					IF eMoverAccessoryID = MoverAccessoryID.APM9001_0000 THEN
						// Note: With the current driver release (3.2209.36.0) mover identification only works if all movers are equiped with ID bumpers!
						bWithBumperID := TRUE;						
					END_IF
				END_FOR
			END_FOR
		END_IF

			
		IF bWithBumperID THEN
			nStatePreparation := nStatePreparation + 10;
		ELSE
			nStatePreparation := 500;
		END_IF
		
	
	60: // 6th: Do mover identification
		//ipVisuMessage.SetInfoMessage('Start mover-identification', 'MoverPreparation', nStatePreparation);
	
		IF NOT bDeterminedMoverID THEN
			IF fbXPlanarSystem.UtilityCheckForError(bAutoReset := TRUE) > 0 THEN
// 				IF fbXPlanarSystem.ipDriver.TcIoXpu(1).SetCoordMoverCommunicationCmd(CoordinatedMoverCommCommand.IdentifyAndAssignPossible) THEN
				IF fbXPlanarSystem.ipDriver.TcIoXpu(1).SetCoordMoverCommunicationCmd(CoordinatedMoverCommCommand.IdentifyBTNsAndRearrangeMovers) THEN
					nStatePreparation := nStatePreparation +1;
				END_IF	
			END_IF
		ELSE
			nStatePreparation := nStatePreparation +10;
		END_IF
	
	61:
		IF fbXPlanarSystem.UtilityCheckForError(bAutoReset := TRUE) > 0 THEN			
			moverCoordComStatus := fbXPlanarSystem.ipDriver.TcIoXpu(1).GetCoordMoverCommStatus();
			
			IF moverCoordComStatus = CoordinatedMoverCommStatus.CommunicationSuccessful THEN
				bDeterminedMoverID := TRUE;
				//ipVisuMessage.ClearAllMessages();
				nStatePreparation := nStatePreparation + 4;
			ELSIF moverCoordComStatus = CoordinatedMoverCommStatus.CommunicationFailed THEN
				nStatePreparation := nStatePreparation + 1;	
			END_IF
			
		END_IF
		
	62:	IF fbXPlanarSystem.UtilityCheckForError(bAutoReset := TRUE) > 0 THEN	
			nMoverID_ErrorCode := fbXPlanarSystem.ipDriver.TcIoXpu(1).GetCoordMoverCommunicationErrorId();
			//ipVisuMessage.SetErrorMessage('Mover Identification Failed!', 'MoverPreparation', nStatePreparation, nMoverID_ErrorCode);
		END_IF
		
		//IF ipVisuMessage.CheckAknowledge()  THEN
		nStatePreparation := 0;	
		//END_IF
	
	65: 
		FOR idx:=1 TO GVL.g_nMoverCount DO
			fbMover[idx].P_MoverID := fbXPlanarSystem.ipDriver.TcIoXpu(1).TcIoMover(UDINT_TO_UINT(idx)).GetIdentifiedMoverBtn();
		END_FOR
		nStatePreparation := nStatePreparation + 5;
	70: // 7th: Determine Mover-Orientation
	
		// Note: At the time of creation of this example code only APM4330 was able to determine its orientation.
		//       Change the code according to newer driver releases and availability of the orientation feature.
		bMoverCanDeterminOrientation := TRUE;
		FOR idx:=1 TO GVL.g_nMoverCount DO
			MoverType := fbXPlanarSystem.ipDriver.TcIoXpu(1).TcIoMover(UDINT_TO_UINT(idx)).GetMoverType();
			IF MoverType <> XPlanarMoverType.APM4330 THEN
				bMoverCanDeterminOrientation := FALSE;
			END_IF
		END_FOR
			
		IF bMoverCanDeterminOrientation THEN
			IF NOT bDerterminedMoverOrientation THEN
				//ipVisuMessage.SetInfoMessage('Mover orientation determination', 'MoverPreparation', nStatePreparation);
				IF fbXPlanarSystem.UtilityCheckForError(bAutoReset := TRUE) > 0 THEN
					IF fbXPlanarSystem.ipDriver.TcIoXpu(1).SetCoordMoverCommunicationCmd(CoordinatedMoverCommCommand.DetermineOrientations) THEN
						nStatePreparation := nStatePreparation + 1;	
					END_IF
				END_IF
			ELSE
				nStatePreparation := nStatePreparation + 20;		
			END_IF
		ELSE
			nStatePreparation := nStatePreparation + 20;
		END_IF
	
		
	71: // Check if communication is active
		IF fbXPlanarSystem.UtilityCheckForError(bAutoReset := TRUE) > 0 THEN
			moverCoordComStatus := fbXPlanarSystem.ipDriver.TcIoXpu(1).GetCoordMoverCommStatus();
			IF moverCoordComStatus = CoordinatedMoverCommStatus.CommunicationInProcess THEN
				nStatePreparation := nStatePreparation + 1;	
			END_IF
		END_IF
	
		
	72: // Wait for orientation determination finished
		IF fbXPlanarSystem.UtilityCheckForError(bAutoReset := TRUE) > 0 THEN
			moverCoordComStatus := fbXPlanarSystem.ipDriver.TcIoXpu(1).GetCoordMoverCommStatus();
			IF moverCoordComStatus = CoordinatedMoverCommStatus.CommunicationSuccessful THEN
				nStatePreparation := nStatePreparation + 8;	
			ELSIF moverCoordComStatus = CoordinatedMoverCommStatus.CommunicationFailed THEN
				IF nCommunicationRetryCounter <= 5 THEN
					nCommunicationRetryCounter := nCommunicationRetryCounter +1;
					nStatePreparation := nStatePreparation - 2;	
				ELSE
					nStatePreparation := nStatePreparation + 1;	
				END_IF
			END_IF
		END_IF
		
				
	73:	// Check which movers do not communicate correctly:
		nMoverToCheck := 0;
		nStatePreparation := nStatePreparation + 1;
		
	74: nMoverToCheck := nMoverToCheck +1;
		IF nMoverToCheck <= GVL.g_nMoverCount THEN
			IF fbXPlanarSystem.UtilityCheckForError(bAutoReset := TRUE) > 0 THEN
				IF fbXPlanarSystem.ipDriver.TcIoXpu(1).TcIoMover(nMoverToCheck).SetMoverCommunicationCommand(MoverCommunicationCommand.DetermineOrientation) THEN
					nStatePreparation := nStatePreparation + 1;
				END_IF
			END_IF
		ELSE
			FOR idx:=1 TO GVL.g_nMoverCount DO
				bCommunicationProblem := FALSE;
				IF bMoverCommunicationProblem[idx] THEN
					bCommunicationProblem := TRUE;	
				END_IF
			END_FOR
			
			IF bCommunicationProblem THEN
				sTextTemp := 'Mover Communication Problem: ';
				FOR idx:=1 TO GVL.g_nMoverCount DO
					IF bMoverCommunicationProblem[idx] THEN
						sTextTemp := CONCAT(sTextTemp, ' M');
						sTextTemp := CONCAT(sTextTemp, UDINT_TO_STRING(idx));
					END_IF
				END_FOR				
				//ipVisuMessage.SetErrorMessage(sTextTemp, sTextTemp, nStatePreparation, 0);
			ELSE
				nStatePreparation := nStatePreparation - 4;	
			END_IF
		END_IF
		
	75: moverComStatus := fbXPlanarSystem.ipDriver.TcIoXpu(1).TcIoMover(nMoverToCheck).GetCommunicationStatus();
		IF moverComStatus = MoverCommunicationStatus.CommunicationSuccessful THEN
			bMoverCommunicationProblem[nMoverToCheck] := FALSE;
			nStatePreparation := nStatePreparation - 1;
		ELSIF moverComStatus = MoverCommunicationStatus.CommunicationFailed THEN
			bMoverCommunicationProblem[nMoverToCheck] := TRUE;
			nStatePreparation := nStatePreparation - 1;
		END_IF
		
		
	80:	// Rotation-Angle modulo adaption
		//ipVisuMessage.SetInfoMessage('Rotation-Angle modulo adaption', 'MoverPreparation', nStatePreparation);
		nMoverToCorrect := 0;
		nStatePreparation := nStatePreparation + 1;	
		
	81:	nMoverToCorrect := nMoverToCorrect +1;
		IF nMoverToCorrect <= GVL.g_nMoverCount THEN
			fMoverOrientationRead    := GVL.g_Movers[nMoverToCorrect].std.P_ActPosition.c; 
			fMoverOrientationCorrect := fMoverOrientationRead;
			 bDoRotationCorrection := FALSE;
			nStatePreparation := nStatePreparation + 1;	
		ELSE
			bDerterminedMoverOrientation := TRUE;
			nStatePreparation := nStatePreparation + 9;	
		END_IF
		
	82:	IF fMoverOrientationCorrect >= 0 THEN
			IF fMoverOrientationCorrect > 360.0 THEN
				fMoverOrientationCorrect := fMoverOrientationCorrect - 180.0;
				bDoRotationCorrection := TRUE;
			ELSE
				nStatePreparation := nStatePreparation + 1;
			END_IF
		ELSE
			IF fMoverOrientationCorrect < 360.0 THEN
				fMoverOrientationCorrect := fMoverOrientationCorrect + 180.0;
				bDoRotationCorrection := TRUE;
			ELSE
				nStatePreparation := nStatePreparation + 1;
			END_IF
		END_IF			
		
		
	83:	IF bDoRotationCorrection THEN
			
			fPosX := GVL.g_Movers[nMoverToCorrect].std.P_ActPosition.x;
			fPosY := GVL.g_Movers[nMoverToCorrect].std.P_ActPosition.y;
			fPosC := GVL.g_Movers[nMoverToCorrect].std.P_ActPosition.c;
	
			CorrectionPos.SetValuesXYC(fPosX, fPosY, fMoverOrientationCorrect);	
	
			GVL.g_Movers[nMoverToCorrect].std.SetMoverPosition('Correction', CorrectionPos);
			
			nStatePreparation := nStatePreparation + 1;	
		ELSE
			nStatePreparation := nStatePreparation - 2;
		END_IF
		
	84:
		IF GVL.g_Movers[nMoverToCorrect].std.P_SetMoverPosition.Done THEN
			nStatePreparation := nStatePreparation - 3;
		ELSIF GVL.g_Movers[nMoverToCorrect].std.P_SetMoverPosition.Error THEN
			nErrorID := GVL.g_Movers[nMoverToCorrect].std.P_SetMoverPosition.ErrorID;
			//ipVisuMessage.SetErrorMessage('Rotation-Angle modulo adaption', 'MoverPreparation', nStatePreparation, nErrorID);		
		END_IF
		

	90: nStatePreparation := 500;
	
			
	500: // Done
	//	nStatePreparation := 0;
		MoverPreparation := TRUE;		
			
		
	END_CASE


	//ipVisuMessage.StateUpdate(nStatePreparation, 'MoverPreparation');
END_METHOD

METHOD MoverRecovery : BOOL
VAR_INPUT
	bReset : BOOL;
END_VAR

VAR
	index : UDINT;
	ipMoverApplication: INT;
END_VAR

VAR_INST
	
	stOptionsJoinTrack				: ST_JoinTrackOptions;
	bMoversJoined 					: BOOL;
	bMoverError 					: BOOL;
	bMoverOrientationSet			: BOOL;
	bClearStation 					:ARRAY [1..GVL.gc_NumberStations] OF BOOL;
	bStationCleared					:bool;
	nMoverToTurn					: UDINT;
	nMoverToTurnBack				: UDINT;
	nTrackToCheck					:UDINT; 
	nDistanceToTrack				:LREAL;
	nDistanceToTargetTrack			: ARRAY[1..moverCount] OF REAL;
	nTargetTrack					: ARRAY[1..moverCount] OF UDINT;
	
	
	
	fRecoveryRotTarget				: LREAL;
	fRecoveryRotVel					: LREAL :=  360.0;
	fRecoveryRotAcc					: LREAL := 1800.0;
	fRecoveryRotJerk				: LREAL := 9000.0;
	stRotationOptions				: ST_MoveCOptions;




	
END_VAR
IF bReset THEN
	MoverRecovery := FALSE;
	nRecoverySequence := 0;
END_IF

CASE nRecoverySequence OF
	0:
		bMoversJoined := FALSE;
		bMoverError := FALSE;
		nMoverToTurn := 0;
		IF NOT bReset THEN
			nRecoverySequence := nRecoverySequence + 1;
		END_IF
		
	1: 	//set rotary orienation 
	
		FOR index := 1 TO gvl.g_nMoverCount DO
		fbXPlanarMover[index].MoveA('', 0, 100, 1000, 1000, 10000);
		fbXPlanarMover[index].MoveB('', 0, 100, 1000, 1000, 10000);
 		fbXPlanarMover[index].MoveC('', 0, 180, 1800, 1800, 18000, 0);
		
		END_FOR

		nRecoverySequence := nRecoverySequence + 1;
	
	2: 
		bMoverOrientationSet:= TRUE; 
		FOR index := 1 TO  gvl.g_nMoverCount DO
			IF fbXPlanarMover[index].P_MoveA.Done AND fbXPlanarMover[index].P_MoveB.Done AND fbXPlanarMover[index].P_MoveC.Done THEN 
				bMoverOrientationSet:= TRUE; 
			ELSE 
				bMoverOrientationSet:= FALSE; 
				
			END_IF
		END_FOR
		
		IF bMoverOrientationSet THEN
			nRecoverySequence := nRecoverySequence + 8;
	
		END_IF
	
	10:
	
		nMoverToTurn := nMoverToTurn +1;
		IF nMoverToTurn > gvl.g_nMoverCount THEN
				nRecoverySequence := nRecoverySequence +3;
			ELSE
				IF GVL.g_Movers[nMoverToTurn].std.P_IsPresent THEN

					fRecoveryRotTarget 				  := GVL.g_Movers[nMoverToTurn].std.P_ClosestQuaterAngle;	
					stRotationOptions.additionalTurns := 0;
					stRotationOptions.direction		  := Tc3_Mc3PlanarMotion.MC_direction.mcDirectionNonModulo;	
					
					GVL.g_Movers[nMoverToTurn].std.MoveC('Recovery - unfinished rotation', fRecoveryRotTarget, fRecoveryRotVel, fRecoveryRotAcc, fRecoveryRotAcc, fRecoveryRotJerk, stRotationOptions);
					nRecoverySequence := nRecoverySequence +1;				
				END_IF	
			END_IF
		
	
	11:
			IF GVL.g_Movers[nMoverToTurn].std.P_MoveC.Done THEN
				nRecoverySequence := nRecoverySequence -1;	
			ELSIF GVL.g_Movers[nMoverToTurn].std.P_MoveC.Error THEN
				nRecoverySequence := nRecoverySequence +1;	
			END_IF
			
	12: 		// Check error ID and react accordingly
			nErrorID := GVL.g_Movers[nMoverToTurn].std.P_MoveC.ErrorID;	
			
			// In case rotation is not possible due to collision with another mover proceed without rotation correction.
			IF nErrorID = 33158 THEN
				nRecoverySequence := nRecoverySequence -2;	
			END_IF

	13: 	nRecoverySequence := 100;	

		    
	100: 
			bStationCleared:=TRUE;
			bClearStation[GVL.PuncherStation]:=fbPuncherStation.Clear();
			bClearStation[GVL.PuncherSeparateStation]:=fbPuncherSeparateStation.Clear();
			bClearStation[GVL.PuncherBufferStation]:=fbPuncherBufferStation.Clear();
	
	FOR  index := 1 TO  GVL.gc_NumberStations DO
		IF bClearStation[index] THEN
			bStationCleared:=TRUE;
			ELSE
				bStationCleared:=FALSE;
		END_IF
	END_FOR
	IF bStationCleared THEN
			nRecoverySequence := 200;

		END_IF
		
// 	110: // look for for nearest track 
// 	
// 	
// 	FOR nMoverToTurnBack := 1 TO  gvl.g_nMoverCount DO
// 		nDistanceToTargetTrack[nMoverToTurnBack]:= 999999;
// 		
// 		FOR nTrackToCheck :=1 TO GVL.gc_NumberTracks DO 
// 		nDistanceToTrack := fbXPlanarMover[ nMoverToTurnBack].GetDistanceToTrack(GVL.g_Tracks[nTrackToCheck].std);
// 		
// 		IF nDistanceToTrack < nDistanceToTargetTrack[nMoverToTurnBack] AND nDistanceToTrack<> -1 THEN 
// 			nDistanceToTargetTrack[nMoverToTurnBack]:=nDistanceToTrack;
// 			nTargetTrack[nMoverToTurnBack] :=nTrackToCheck;
// 		END_IF
// 		
// 	END_FOR
// 	
// 	END_FOR
// 	
// 	nRecoverySequence := nRecoverySequence +10;
// 	
// 	120: // join to track
// 
// 		stOptionsJoinTrack.useOrientation := TRUE;
// 		
// 		FOR index := 1 TO gvl.g_nMoverCount DO
// 		IF fbXPlanarMover[index].P_CommandMode<> MC_PLANAR_MOVER_COMMAND_MODE.OnTrack THEN
// 			fbXPlanarMover[index].JoinTrack('Joining track', GVL.g_Tracks[nTargetTrack[index]].std, 250, 1250, 12500, stOptionsJoinTrack);
// 			
// 		END_IF
// 		
// 			
// END_FOR
// 	
// 		nRecoverySequence := nRecoverySequence + 1;
// 		
// 	121:
// 		bMoversJoined := TRUE;
// 		bMoverError := FALSE;
// 		FOR index := 1 TO moverCount DO
// 			bMoversJoined := bMoversJoined AND fbXPlanarMover[index].P_JoinTrack.Done;
// 			IF  fbXPlanarMover[index].P_JoinTrack.Done THEN 
// 				gvl.g_Movers[index].P_TrackId:=nTargetTrack[index];
// 			END_IF
// 			bMoverError := bMoverError OR fbXPlanarMover[index].P_JoinTrack.Error;			
// 		END_FOR
// 		
// 	IF bMoversJoined THEN
// 			nRecoverySequence := nRecoverySequence + 9;
// 	ELSIF bMoverError THEN
//  			nRecoverySequence := nRecoverySequence + 4;
// 	END_IF
// 		
		
// 	130: //send mover to station 
// 	  	  
// 		FOR index := 1 TO gvl.g_nMoverCount DO
// 			 IF fbXPlanarMover[index].P_TrackId= GVL.TrackPuncherWellplate THEN 
// 				 fbPuncherStation.P_List_Switch_Input_W.AddMover(GVL.g_Movers[index].std);
// 		
// 			
// 			 END_IF
// 		END_FOR
// 
// 		nRecoverySequence := 200;

	200: 
		MoverRecovery := TRUE;
		
END_CASE
END_METHOD

METHOD Resetting : BOOL
VAR_INPUT
END_VAR

VAR
	index : UDINT;
	MC_PLANNAR_: ST_CommandReturn;
END_VAR


VAR_INST
	
	nTrackToEnable		: UDINT;
	stProductDataClear 	: ST_ProductData;
	stOptionsJoinTrack				: ST_JoinTrackOptions;
	bMoversJoined 					: BOOL;
	bMoverError 					: BOOL;
	nMoverToTurn					: UDINT;
	nMoverToTurnBack				: UDINT;
	nTrackToCheck					:UDINT; 
	nDistanceToTrack				:LREAL;
	nDistanceToTargetTrack			: ARRAY[1..moverCount] OF REAL;
	nTargetTrack					: ARRAY[1..moverCount] OF UDINT;
	
END_VAR
nErrorID := 0;

CASE nResettingSequence OF 
	
	0: // Enter 
		nResettingSequence := 10;
		
		
		
	10: // Reset all movers
		IF fbXPlanarSystem.ResetMovers() THEN
		//	ipVisuMessage.SetInfoMessage('RESET all movers', 'Resetting', nResettingSequence);
			nResettingSequence := nResettingSequence +1;			
		END_IF
		
	11: IF fbXPlanarSystem.P_ResetMovers.Done THEN
			nResettingSequence := nResettingSequence +9;
		ELSIF fbXPlanarSystem.P_ResetMovers.Error THEN
			nResettingSequence := nResettingSequence +1;	
		END_IF

	12:	// Check error ID and react accordingly
		nErrorID := fbXPlanarSystem.P_EnableMovers.ErrorID;
		//ipVisuMessage.SetErrorMessage('RESET movers failed', 'Resetting', nResettingSequence, nErrorID);					
		
		
		
	20:	// Reset all tracks
		IF fbXPlanarSystem.ResetTracks() THEN
			//ipVisuMessage.SetInfoMessage('RESET all tracks', 'Resetting', nResettingSequence);
			nResettingSequence := nResettingSequence +1;
		END_IF
		
	21: IF fbXPlanarSystem.P_ResetTracks.Done THEN
			nResettingSequence := nResettingSequence +19;
	 	ELSIF fbXPlanarSystem.P_ResetTracks.Error THEN
			nResettingSequence := nResettingSequence +1;	
		END_IF
	
	22:	// Check error ID and react accordingly
		nErrorID := fbXPlanarSystem.P_EnableMovers.ErrorID;
		//ipVisuMessage.SetErrorMessage('RESET tracks failed', 'Resetting', nResettingSequence, nErrorID);			
		
	
		
// 	30:	// Reset MotionSystemApplication
// 		IF ipMotionSystemApplication.Reset() THEN
// 		//	ipVisuMessage.SetInfoMessage('RESET MotionSystemApplication', 'Resetting', nResettingSequence);
// 			nResettingSequence := nResettingSequence +10;
// 		END_IF
	
				
	40:  // Cleaning all process data
		FOR idx:=1 TO GVL.g_nMoverCount DO
		//	ipMoverApplication[idx].P_ProductData := stProductDataClear;
		END_FOR
		nResettingSequence := nResettingSequence+10;
		
	50: // check if any mover is disable 
			
		FOR index := 1 TO gvl.g_nMoverCount DO
			 IF fbXPlanarMover[index].P_State=MC_PLANAR_STATE.Disabled THEN 
				 nResettingSequence := nResettingSequence + 1;
				 RETURN; 
			 END_IF
		END_FOR
			 nResettingSequence :=100;
	 
	51:	// enable movers
			IF fbXPlanarSystem.EnableMovers() THEN
				nResettingSequence := nResettingSequence + 1;
			END_IF
	
	52: // wait for enabling
		IF fbXPlanarSystem.P_EnableMovers.Done THEN
			nResettingSequence := 100;
		ELSIF fbXPlanarSystem.P_EnableMovers.Error THEN
			nResettingSequence := nResettingSequence + 3;
			nErrorID := fbXPlanarSystem.P_EnableMovers.ErrorID;
 		END_IF
		
// 	60:  // look for for nearest track 
// 	
// 		FOR nMoverToTurnBack := 1 TO  gvl.g_nMoverCount DO
// 			nDistanceToTargetTrack[nMoverToTurnBack]:= 999999;
// 			
// 			FOR nTrackToCheck :=1 TO 10 DO//GVL.gc_NumberTracks DO 
// 			nDistanceToTrack := fbXPlanarMover[ nMoverToTurnBack].GetDistanceToTrack(GVL.g_Tracks[nTrackToCheck].std);
// 			
// 				IF nDistanceToTrack < nDistanceToTargetTrack[nMoverToTurnBack] THEN 
// 					nDistanceToTargetTrack[nMoverToTurnBack]:=nDistanceToTrack;
// 					nTargetTrack[nMoverToTurnBack] :=nTrackToCheck;
// 				END_IF
// 			
// 			END_FOR
// 	
// 		END_FOR
// 		
// 	nResettingSequence := nResettingSequence +10;
// 	
// 	70: // join to track
// 
// 		stOptionsJoinTrack.useOrientation := TRUE;
// 		
// 		FOR index := 1 TO gvl.g_nMoverCount DO
// 		IF fbXPlanarMover[index].P_CommandMode<> MC_PLANAR_MOVER_COMMAND_MODE.OnTrack THEN
// 			fbXPlanarMover[index].JoinTrack('Joining track', GVL.g_Tracks[nTargetTrack[index]].std, 250, 1250, 12500, stOptionsJoinTrack);
// 			END_IF
// 
// END_FOR
// 	
// 		nResettingSequence := nResettingSequence + 1;
// 		
// 	71:
// 		bMoversJoined := TRUE;
// 		bMoverError := FALSE;
// 		FOR index := 1 TO moverCount DO
// 			bMoversJoined := bMoversJoined AND fbXPlanarMover[index].P_JoinTrack.Done;
// 			bMoverError := bMoverError OR fbXPlanarMover[index].P_JoinTrack.Error;			
// 		END_FOR
// 		
// 	IF bMoversJoined THEN
// 			nResettingSequence := 100;
// 	ELSIF bMoverError THEN
//  			nResettingSequence := nResettingSequence + 4;
// 	END_IF
// 		
	
	100: // Reset done
		//ipVisuMessage.SetInfoMessage('RESET finished', 'Resetting', 0);
	
		nResettingSequence := 0; 
		         Resetting := TRUE;

END_CASE



//ipVisuMessage.StateUpdate(nResettingSequence, 'Resetting');
END_METHOD

METHOD Starting : BOOL
VAR_INPUT
	bReset : BOOL;
END_VAR

VAR 
	nErrorID : UDINT;
	nMoverIndex: UDINT;
END_VAR
IF bReset THEN
	Starting := FALSE;
	nStartingSequence := 0;
END_IF

CASE nStartingSequence OF
	0: //init
		Execute(bReset := TRUE);
		MoverRecovery(bReset := TRUE);
		IF NOT bReset THEN
			nStartingSequence := nStartingSequence + 10;
		END_IF
	10: // enable collision avoidance group
		IF fbXPlanarSystem.EnableGroup() THEN
			nStartingSequence := nStartingSequence + 1;
		END_IF
	11:
		IF fbXPlanarSystem.P_EnableGroup.Done THEN
			nStartingSequence := nStartingSequence + 9;
		ELSIF fbXPlanarSystem.P_EnableGroup.Error THEN
			nStartingSequence := nStartingSequence + 4;
			nErrorID := fbXPlanarSystem.P_EnableGroup.ErrorID;
		END_IF
	20: // add environment 
		IF fbXPlanarSystem.AddEnvironmentToGroup() THEN
			nStartingSequence := nStartingSequence + 1;
		END_IF
	21: 
		IF fbXPlanarSystem.P_AddEnviromentToGroup.Done THEN
			nStartingSequence := nStartingSequence + 9;
		ELSIF fbXPlanarSystem.P_AddEnviromentToGroup.Error THEN
			nStartingSequence := nStartingSequence + 4;
			nErrorID := fbXPlanarSystem.P_AddEnviromentToGroup.ErrorID;
		END_IF
		
	30:
		IF fbXPlanarSystem.EnableTracks() THEN
			nStartingSequence := nStartingSequence + 1;
		END_IF
	
	31: 
		IF fbXPlanarSystem.P_EnableTracks.Done THEN
			nStartingSequence := nStartingSequence + 9;
		ELSIF fbXPlanarSystem.P_EnableTracks.Error THEN
			nStartingSequence := nStartingSequence + 4;
			nErrorID := fbXPlanarSystem.P_EnableTracks.ErrorID;
		END_IF
	
			
	40:
		IF fbXPlanarSystem.AddTracksToGroup() THEN
			nStartingSequence := nStartingSequence + 1;
		END_IF
	
	41: 
		IF fbXPlanarSystem.P_AddTracksToGroup.Done THEN
			nStartingSequence := nStartingSequence + 1;
		ELSIF fbXPlanarSystem.P_AddTracksToGroup.Error THEN
			nStartingSequence := nStartingSequence + 4;
			nErrorID := fbXPlanarSystem.P_AddTracksToGroup.ErrorID;
		END_IF
		
	42: // Prepare all movers
		IF MoverPreparation(bReset:=TRUE) THEN
			nStartingSequence := nStartingSequence + 1;
		END_IF
		
	43:
		IF MoverPreparation(bReset:=FALSE) THEN
			nStartingSequence := nStartingSequence + 7;
		END_IF	
		
	50: // enable movers
		IF fbXPlanarSystem.EnableMovers() THEN
			nStartingSequence := nStartingSequence + 1;
		END_IF
	51: // wait for enabling
		IF fbXPlanarSystem.P_EnableMovers.Done THEN
			nStartingSequence := nStartingSequence + 9;
		ELSIF fbXPlanarSystem.P_EnableMovers.Error THEN
			nStartingSequence := nStartingSequence + 4;
			nErrorID := fbXPlanarSystem.P_EnableMovers.ErrorID;
		END_IF
	60: // add movers to group
		IF fbXPlanarSystem.AddMoversToGroup() THEN
			nStartingSequence := nStartingSequence + 1;
		END_IF
	61: // wait for enabling
		IF fbXPlanarSystem.P_AddMoversToGroup.Done THEN
			nStartingSequence := nStartingSequence + 1;
		ELSIF fbXPlanarSystem.P_AddMoversToGroup.Error THEN
			nStartingSequence := nStartingSequence + 4;
			nErrorID := fbXPlanarSystem.P_AddMoversToGroup.ErrorID;
		END_IF
	62:
	 	FOR nMoverIndex := 1 TO GVL.g_nMoverCount DO
			GVL.g_Movers[nMoverIndex].std.P_Id := UDINT_TO_UINT(nMoverIndex);
		END_FOR
		nStartingSequence := nStartingSequence + 8;
	70:
		IF MoverRecovery(bReset := FALSE) THEN
			nStartingSequence := nStartingSequence + 10;
		END_IF
	80: 
		Starting := TRUE;
END_CASE
END_METHOD

METHOD Startup : BOOL
VAR_INPUT
END_VAR

VAR
	index : UDINT;
		stMoverDetectionInfos   : ST_TcIoMoverDetectionInfos;
		detectedMovers:UDINT; 
END_VAR

VAR_INST
	aTrackTable : ARRAY[1..maxTrackCount] OF FB_TrackTable;
	nTrackIdx: UDINT;
	nStationToInit : UINT;
	
	nStartFromTrack : UDINT;
	nEndAtTrack : UDINT;
	bCloseLoop : BOOL;
END_VAR
CASE nStartupSequence OF
	0: //init
		nStartupSequence := nStartupsequence + 1;
		bAssignmentComplete := FALSE;
	
	1: //assign mover to system
		
		FOR index := 1 TO MoverCount DO
			fbMover[index].std := THIS^.fbXPlanarMover[index];
		END_FOR	
		//nStartupSequence := nStartupSequence + 1;
	
		FOR index := 1 TO moverCount DO
			fbXPlanarSystem.SetMoverStandard(index, THIS^.fbXPlanarMover[index]);
		END_FOR
		
		nStartupSequence := nStartupSequence + 1;
		
	2:  // Movers to global mover interface
		FOR index := 1 TO MoverCount DO
			GVL.g_Movers[index] := THIS^.fbMover[index];
			THIS^.fbMover[index].P_MoverIndex := UDINT_TO_INT(index); 
		END_FOR	
		nStartupSequence := nStartupSequence + 1;
	
	3:  // Assigning global Track-Interfaces
		GVL.g_Tracks[GVL.TrackPuncherWellplate] := THIS^.fbTrackPuncherWellplate;
		GVL.g_Tracks[GVL.TrackBufferPuncher] := THIS^.fbTrackBufferPuncher;
		GVL.g_Tracks[GVL.TrackStradeFirstSeg] := THIS^.fbTrackStradeFirstSeg;
		GVL.g_Tracks[GVL.TrackStradeSecondSeg] := THIS^.fbTrackStradeSecondSeg;
		GVL.g_Tracks[GVL.TrackPipettePreBuffer] := THIS^.fbTrackPipettePreBuffer;
		GVL.g_Tracks[GVL.TrackPipette] := THIS^.fbTrackPipette;
		GVL.g_Tracks[GVL.TrackPipettePostBuffer] := THIS^.fbTrackPipettePostBuffer;
		GVL.g_Tracks[GVL.TrackPipetteBufferCon] := THIS^.fbTrackPipetteBufferCon;
		GVL.g_Tracks[GVL.TrackUserInteraction] := THIS^.fbTrackUserInteraction;
		GVL.g_Tracks[GVL.CloseLoopTrack] := THIS^.fbCloseLoopTrack;
		GVL.g_Tracks[GVL.PuncherSeperateTrack] := THIS^.fbPuncherSeperate;
		
		
		nTrackIdx := 0;
		bAssignmentComplete := TRUE;
		nStartupSequence := nStartupSequence + 1;	
		
	4: //assign track to system
		FOR index := 1 TO GVL.gc_NumberTracks DO
			fbXPlanarSystem.SetTrackStandard(index, GVL.g_Tracks[index].std);
		END_FOR
		
		nStartupSequence := nStartupSequence + 1;
	
	5: // assign stations
		GVL.g_Stations[GVL.PuncherStation] := THIS^.fbPuncherStation;
		GVL.g_Stations[GVL.PuncherSeparateStation] := THIS^.fbPuncherSeparateStation;
		GVL.g_Stations[GVL.PuncherBufferStation] := THIS^.fbPuncherBufferStation;
		
		nStartupSequence := nStartupSequence + 6;
		
	11: // Track number count
		IF nTrackIdx < GVL.gc_NumberTracks THEN
			nTrackIdx := nTrackIdx + 1;
			nStartupSequence := nStartupSequence +1;
		ELSE
			    nTrackIdx := 0;
			nStartupSequence := 14;
		END_IF
				
	12:	// Clear track data
		IF GVL.g_Tracks[nTrackIdx].Clear() THEN
			nStartupSequence := nStartupSequence +1;
		END_IF
		
	13: // Build the track
		IF GVL.g_Tracks[nTrackIdx].Initialize(nTrackIdx) THEN	
			nStartupSequence := 11;
		ELSE
			IF GVL.g_Tracks[nTrackIdx].P_Error THEN
				nStartupSequence := nStartupSequence +1;
			END_IF
		END_IF
		
	14: // Init all stations
		nStationToInit := 0;
		nStartupSequence := nStartupSequence +1;

	15:	nStationToInit := nStationToInit +1;
		IF nStationToInit <= GVL.gc_NumberStations THEN
			nStartupSequence := nStartupSequence +1;
		ELSE
			nStartupSequence := 30;
		END_IF	
				
	16: IF GVL.g_Stations[nStationToInit].Init() THEN
			nStartupSequence := nStartupSequence -1;
		END_IF

	30: 
		Startup := TRUE;
END_CASE
END_METHOD

END_FUNCTION_BLOCK

// ---- Tracks/FB_PuncherWellplateTrack.TcPOU
FUNCTION_BLOCK FB_PuncherWellplateTrack EXTENDS FB_BaseTrack implements I_Track;
VAR_INPUT
END_VAR
VAR_OUTPUT
END_VAR
VAR
END_VAR

METHOD Initialize : BOOL
VAR_INPUT
	nTrackIndex	: UDINT;
END_VAR

VAR_INST
	TrackTable		: FB_TrackTable;
	
	bIsDone : BOOL;
	bIsActive : BOOL;
	bIsError : BOOL;
	stRet : ST_CommandReturn;
END_VAR


CASE nInitState OF
	10:	// Starting with an empty table. 
		IF TrackTable.ClearTrackTable() THEN
			nInitState := nInitState + 10;
		END_IF
	20: 
		// Init Track-Table
		
		// *************************************************************************************
		// *** Only the code in this state must be eddited according to machine/track layout ***
		// *************************************************************************************	
		
		nStartFromTrack	:= 0;		// 0 for the first track all others according to their predecessor!
	    	nEndAtTrack := 0;		// 0 for the first track all others according to their successor! 		
		     bCloseLoop := FALSE;	// TRUE for circular track	
		
		TrackTable.AddPoint(E_PointType.Line_Start, E_PointOption.none, 600, 60, 0);
		TrackTable.AddPoint(E_PointType.Line_End, E_PointOption.none, 550, 60, 0);
		
		TrackTable.AddPoint(E_PointType.Line_Start, E_PointOption.none, 540, 70, 0);
		TrackTable.AddPoint(E_PointType.Line_End, E_PointOption.none, 540, 290, 0);
		
		nInitState := nInitState + 10;
		
	30:
		// *************************************************************
		// ***       NO Code Changes are needed from here on!        ***
		// *************************************************************		
			
		// The track table contains all additional information, too.
		IF nStartFromTrack > 0 THEN
			TrackTable.P_StartFromTrack := GVL.g_Tracks[nStartFromTrack].std;	
		END_IF
		IF nEndAtTrack > 0 THEN
			TrackTable.P_EndAtTrack := GVL.g_Tracks[nEndAtTrack].std;	
		END_IF	
		TrackTable.P_CloseTheLoop := bCloseLoop;	
		nInitState := nInitState + 10;

			
		
	40: // Checking the track table for plausibility
		IF TrackTable.CheckTrackTable() <> 0 THEN
			IF TrackTable.P_TrackTableCheckResult THEN
				nInitState := 50;	// Plausibility test succeeded.
			ELSE
				nInitState := 41;	// Plausibility test failed!
			END_IF
		END_IF
	41:	// In case of failed plausibility test check the creation of the above track table.
		// A Line must always begin with E_PointType.Line_Start and end with E_PointType.Line_End.
		// A Circle must always be added in the order E_PointType.Circle_Start, E_PointType.Circle_Center, E_PointType.Circle_End.
		// Check the info text for further information:
		bTrackBuildError := TRUE;
							
 					   
	50:	// Building the track	
		IF fbTrackStandard.BuildTrackExt(TrackTable) THEN
			nInitState := nInitState +1;
		END_IF
		
	51:	
		bIsDone := fbTrackStandard.P_BuildTrackExt.Done;
		bIsActive := fbTrackStandard.P_BuildTrackExt.Active;
		bIsError := fbTrackStandard.P_BuildTrackExt.Error;
		stRet := fbTrackStandard.P_BuildTrackExt;
		
		IF fbTrackStandard.P_BuildTrackExt.Done THEN
			nInitState := 100;	
		ELSIF fbTrackStandard.P_BuildTrackExt.Error THEN
	  		nInitState := nInitState +1;
		END_IF		
		
	52: // In case an error occured, check the error ID and InfoText and react accordingly:
		   bTrackBuildError := TRUE;
		 
	100: 	// Track build done
			fTrackLength := fbTrackStandard.GetLength();
			  Initialize := TRUE;
	
			
END_CASE
END_METHOD

PROPERTY P_Error : Bool
GET
P_Error := bTrackBuildError;
END_GET
END_PROPERTY

END_FUNCTION_BLOCK

// ---- Tracks/FB_StradeFirstSegTrack.TcPOU
FUNCTION_BLOCK FB_StradeFirstSegTrack EXTENDS FB_BaseTrack implements I_Track;
VAR_INPUT
END_VAR
VAR_OUTPUT
END_VAR
VAR
END_VAR

METHOD Initialize : BOOL
VAR_INPUT
	nTrackIndex	: UDINT;
END_VAR

VAR_INST
	TrackTable		: FB_TrackTable;
	
	bIsDone : BOOL;
	bIsActive : BOOL;
	bIsError : BOOL;
	stRet : ST_CommandReturn;
END_VAR


CASE nInitState OF
	10:	// Starting with an empty table. 
		IF TrackTable.ClearTrackTable() THEN
			nInitState := nInitState + 10;
		END_IF
	20: 
		// Init Track-Table
		
		// *************************************************************************************
		// *** Only the code in this state must be eddited according to machine/track layout ***
		// *************************************************************************************	
		
		nStartFromTrack	:= 1;		// 0 for the first track all others according to their predecessor!
	    	nEndAtTrack := 0;		// 0 for the first track all others according to their successor! 		
		     bCloseLoop := FALSE;	// TRUE for circular track	

		TrackTable.AddPoint(E_PointType.Line_Start, E_PointOption.none, 530, 300, 0);
		TrackTable.AddPoint(E_PointType.Line_End, E_PointOption.none, 360, 300, 0);
		
		nInitState := nInitState + 10;
		
	30:
		// *************************************************************
		// ***       NO Code Changes are needed from here on!        ***
		// *************************************************************		
			
		// The track table contains all additional information, too.
		IF nStartFromTrack > 0 THEN
			TrackTable.P_StartFromTrack := GVL.g_Tracks[nStartFromTrack].std;	
		END_IF
		IF nEndAtTrack > 0 THEN
			TrackTable.P_EndAtTrack := GVL.g_Tracks[nEndAtTrack].std;	
		END_IF	
		TrackTable.P_CloseTheLoop := bCloseLoop;	
		nInitState := nInitState + 10;

			
		
	40: // Checking the track table for plausibility
		IF TrackTable.CheckTrackTable() <> 0 THEN
			IF TrackTable.P_TrackTableCheckResult THEN
				nInitState := 50;	// Plausibility test succeeded.
			ELSE
				nInitState := 41;	// Plausibility test failed!
			END_IF
		END_IF
	41:	// In case of failed plausibility test check the creation of the above track table.
		// A Line must always begin with E_PointType.Line_Start and end with E_PointType.Line_End.
		// A Circle must always be added in the order E_PointType.Circle_Start, E_PointType.Circle_Center, E_PointType.Circle_End.
		// Check the info text for further information:
		bTrackBuildError := TRUE;
							
 					   
	50:	// Building the track	
		IF fbTrackStandard.BuildTrackExt(TrackTable) THEN
			nInitState := nInitState +1;
		END_IF
		
	51:	
		bIsDone := fbTrackStandard.P_BuildTrackExt.Done;
		bIsActive := fbTrackStandard.P_BuildTrackExt.Active;
		bIsError := fbTrackStandard.P_BuildTrackExt.Error;
		stRet := fbTrackStandard.P_BuildTrackExt;
		
		IF fbTrackStandard.P_BuildTrackExt.Done THEN
			nInitState := 100;	
		ELSIF fbTrackStandard.P_BuildTrackExt.Error THEN
	  		nInitState := nInitState +1;
		END_IF		
		
	52: // In case an error occured, check the error ID and InfoText and react accordingly:
		   bTrackBuildError := TRUE;
		 
	100: 	// Track build done
			fTrackLength := fbTrackStandard.GetLength();
			  Initialize := TRUE;
	
			
END_CASE
END_METHOD

PROPERTY P_Error : Bool
GET
P_Error := bTrackBuildError;
END_GET
END_PROPERTY

END_FUNCTION_BLOCK

// ---- Tracks/FB_PipettePostBufferTrack.TcPOU
FUNCTION_BLOCK FB_PipettePostBufferTrack EXTENDS FB_BaseTrack implements I_Track;
VAR_INPUT
END_VAR
VAR_OUTPUT
END_VAR
VAR
END_VAR

METHOD Initialize : BOOL
VAR_INPUT
	nTrackIndex	: UDINT;
END_VAR

VAR_INST
	TrackTable		: FB_TrackTable;
	
	bIsDone : BOOL;
	bIsActive : BOOL;
	bIsError : BOOL;
	stRet : ST_CommandReturn;
END_VAR


CASE nInitState OF
	10:	// Starting with an empty table. 
		IF TrackTable.ClearTrackTable() THEN
			nInitState := nInitState + 10;
		END_IF
	20: 
		// Init Track-Table
		
		// *************************************************************************************
		// *** Only the code in this state must be eddited according to machine/track layout ***
		// *************************************************************************************	
		
		nStartFromTrack	:= 6;		// 0 for the first track all others according to their predecessor!
	    	nEndAtTrack := 0;		// 0 for the first track all others according to their successor! 		
		     bCloseLoop := FALSE;	// TRUE for circular track	
		
		TrackTable.AddPoint(E_PointType.Line_Start, E_PointOption.none, 110, 60, 0);
		TrackTable.AddPoint(E_PointType.Line_End, E_PointOption.none, 60.01, 60, 0);
		
		TrackTable.AddPoint(E_PointType.Line_Start, E_PointOption.none, 60, 60.01, 0);
		TrackTable.AddPoint(E_PointType.Line_End, E_PointOption.none, 60, 299.99, 0);
		
		nInitState := nInitState + 10;
		
	30:
		// *************************************************************
		// ***       NO Code Changes are needed from here on!        ***
		// *************************************************************		
			
		// The track table contains all additional information, too.
		IF nStartFromTrack > 0 THEN
			TrackTable.P_StartFromTrack := GVL.g_Tracks[nStartFromTrack].std;	
		END_IF
		IF nEndAtTrack > 0 THEN
			TrackTable.P_EndAtTrack := GVL.g_Tracks[nEndAtTrack].std;	
		END_IF	
		TrackTable.P_CloseTheLoop := bCloseLoop;	
		nInitState := nInitState + 10;

			
		
	40: // Checking the track table for plausibility
		IF TrackTable.CheckTrackTable() <> 0 THEN
			IF TrackTable.P_TrackTableCheckResult THEN
				nInitState := 50;	// Plausibility test succeeded.
			ELSE
				nInitState := 41;	// Plausibility test failed!
			END_IF
		END_IF
	41:	// In case of failed plausibility test check the creation of the above track table.
		// A Line must always begin with E_PointType.Line_Start and end with E_PointType.Line_End.
		// A Circle must always be added in the order E_PointType.Circle_Start, E_PointType.Circle_Center, E_PointType.Circle_End.
		// Check the info text for further information:
		bTrackBuildError := TRUE;
							
 					   
	50:	// Building the track	
		IF fbTrackStandard.BuildTrackExt(TrackTable) THEN
			nInitState := nInitState +1;
		END_IF
		
	51:	
		bIsDone := fbTrackStandard.P_BuildTrackExt.Done;
		bIsActive := fbTrackStandard.P_BuildTrackExt.Active;
		bIsError := fbTrackStandard.P_BuildTrackExt.Error;
		stRet := fbTrackStandard.P_BuildTrackExt;
		
		IF fbTrackStandard.P_BuildTrackExt.Done THEN
			nInitState := 100;	
		ELSIF fbTrackStandard.P_BuildTrackExt.Error THEN
	  		nInitState := nInitState +1;
		END_IF		
		
	52: // In case an error occured, check the error ID and InfoText and react accordingly:
		   bTrackBuildError := TRUE;
		 
	100: 	// Track build done
			fTrackLength := fbTrackStandard.GetLength();
			  Initialize := TRUE;
	
			
END_CASE
END_METHOD

PROPERTY P_Error : Bool
GET
P_Error := bTrackBuildError;
END_GET
END_PROPERTY

END_FUNCTION_BLOCK

// ---- Stations/FB_PuncherSeparateStation.TcPOU
FUNCTION_BLOCK FB_PuncherSeparateStation EXTENDS FB_StationBase

METHOD Clear : BOOL
	CASE nStateClear OF
		
	0:	// Enter
		Clear := FALSE;
		nStateClear := nStateClear +10;
		
	10: // Clearing all Station-Lists 
		IF SUPER^.Clear() THEN
			nStateClear := nStateClear +10;
		END_IF	
	
	20:	// Add aditional Data to be cleared here...
		nStateClear := 100;
		
		
	100: // Done
		      Clear := TRUE;
		nStateClear := 0;

	END_CASE
END_METHOD

METHOD Init : BOOL


VAR_INST
	nTestCounter	: INT;	
END_VAR
nTestCounter := nTestCounter +1;

CASE nStateInit OF

	0:		// Enter 
			bStationInitDone := FALSE;
			   nStateProcess := 0;
			      nStateInit := 10;
				 
			
	10:		// Init Station-Parameters				
				  nStationIndex := 2;				// Each station needs an unique index	
			 nStationTrackIndex := 11;	 			// Track on which the station resides
			 
	nPreviousStationIndexInputN := 0;
			  nTrackIndexInputN := 0;
	   nNextStationIndexOutputN := 0;
	   		 nTrackIndexOutputN := 0;
			 

			 fStationPosition_X := 663.0;			// Position of the station in X/Y coordinates
			 fStationPosition_Y := 238.0;			// Position of the station in X/Y coordinates
			  
	   fSendAwayDistanceOutputN := 0.0;			// Position on track a mover will be send to after processing 
	  							// Position on track a mover will be send to after processing 
			  fInRangeDistance  := 300.0;			// Position in front of a station from where a mover will be taken over
			  
			  nStateInit := 11;
				   
				  
	11: // Fail-safe check, just to make sure all variables have been assigned after doing copy&paste from the template
			IF        nStationIndex > 0
			AND  nStationTrackIndex > 0
			AND  fStationPosition_X > 0
			AND  fStationPosition_Y > 0
			AND   fInRangeDistance > 0
			THEN   
				nStateInit := 20;
			END_IF
			
				   
	20:		// Calculating positions
	
			// 1. Calculating station position on track
			position.SetValuesXYC(fStationPosition_X, fStationPosition_Y, 0.0);
			//fStationPositionOnTrack := GVL.g_Tracks[nStationTrackIndex].std.GetTrackPositionAt_XY(fStationPosition_X, fStationPosition_Y);
			fStationPositionOnTrack := GVL.g_Tracks[nStationTrackIndex].P_TrackLength;				
			
			// 2. Calculating send-away position on track
// 			fSendAwayPositionOutputS := fStationPositionOnTrack + fSendAwayDistanceOutputS; 
// 			fSendAwayPositionOutputE := fSendAwayDistanceOutputE; 
// 		
// 			// The send away position must not exceed the lenght of the following track!
// 			fSendAwayPositionOutputS := MIN(MAX(0, fSendAwayPositionOutputS), GVL.g_Tracks[nTrackIndexOutputS].P_TrackLength);
// 			fSendAwayPositionOutputE := MIN(MAX(0, fSendAwayPositionOutputE), GVL.g_Tracks[nTrackIndexOutputE].P_TrackLength);
// 			
			// 3. Calculating the station position in X/Y coordinates determined by the track	
            //    This is to make sure the center of the station is always located directly on the track.
			//    This value can differ from the initial fStationPosition_X, fStationPosition_Y in case they were not matching the track
			GVL.g_Tracks[nStationTrackIndex].std.GetMoverPositionAt(fStationPositionOnTrack, StationPosition);
			
			// Providing the station position to e.g. visualization	
			stStationPosition.bInit            := TRUE;
			stStationPosition.fPositionOnTrack := fStationPositionOnTrack;
			stStationPosition.nTrackId         := nStationTrackIndex;
			stStationPosition.fPosition_X	   := StationPosition.x;
			stStationPosition.fPosition_Y	   := StationPosition.y;

			nStateInit := 30;
			
			
	30:		// Clear Lists
			IF THIS^.Clear() THEN
				nStateInit := 90;	
			END_IF

			
		
	90:		// Creating a little history of what happened in the station for debugging purpose
			fbHistoryInfo.AddEntry('Init');
	
			nStateInit := 100;
			
						
	100:	// Init done
			IF SUPER^.Init() THEN
				bStationInitDone := TRUE;	
				           Init := TRUE;
			END_IF
				
	
END_CASE
END_METHOD

METHOD Process : BOOL

VAR_INST
		
	nMoverIndex				: UINT;
	
	fMoverToTrackPosition	: LREAL;
	nTrackIndex				: UINT;
	fMoverVelocity			: LREAL;
	fMoverAcceleration		: LREAL;
	fMoverJerk				: LREAL;
	
	
	nErrorId				: UDINT;
	nObjectID				: UDINT;
	nObjectType				: UDINT;		
	
	
	// Process
	nDestinationProcess		: UINT;
	nIncommingTrackOID		: UDINT;
	nNextStationIndex		: UINT;		 				
	fSendAwayPosition		: LREAL;
	nTrackindexNext			: UINT;

	// positions
	loadPosition 			: PositionXYC;
	rotatePosition 			: PositionXYC;
	unloadPosition 			: PositionXYC;
	
	//movemets setup
	stMoveToPositionOptions: ST_MoveToPositionOptions;


END_VAR


VAR
	bPartInGripper: BOOL; 
	ipMoverApplication: INT;
END_VAR
// Station - Switch-Seperate

CASE nStateProcess OF 

	0:		// Enter
			IF bStationInitDone THEN
				nStateProcess := 100;
			END_IF

	
	100: 	// Waiting for Mover
			IF P_List_Switch_Input_N.P_FirstInList <> 0 THEN
				P_List_Station.AddMover(P_List_Switch_Input_N.RemoveFirstInList());
			    nStateProcess := nStateProcess +10;
			END_IF
	
			
	110:	// Working with the station list from here on	
			IF P_List_Station.P_FirstInList <> 0 THEN
				nMoverIndex := P_List_Station.P_FirstInList.P_Id;
			    nStateProcess := nStateProcess +10;
			END_IF		
			
			
	120: 	// Check if Mover is in range
			IF    GVL.g_Movers[nMoverIndex].std.P_SetOnTrack.TrackOID = GVL.g_Tracks[nTrackIndexInputN].std.P_OID
			AND   GVL.g_Movers[nMoverIndex].std.P_SetOnTrack.SetPos   > fStationPositionOnTrack - fInRangeDistance
			THEN
				nStateProcess := nStateProcess +10;
			END_IF
			
			
			

			
			
		
	130: 	// Send mover to the track position 
			fSendAwayPosition		:=0;	
			fMoverToTrackPosition := fSendAwayPosition;
			nTrackIndex           := nStationTrackIndex;
			fMoverVelocity     	  :=    300.0;
			fMoverAcceleration 	  :=  1_000.0;
			fMoverJerk         	  := 10_000.0;	
	
			stMoveOnTrackParameters.direction := Tc3_Mc3PlanarMotion.MC_DIRECTION.mcDirectionShortestWay;	
			stMoveOnTrackParameters.gap := 120.0;

			
			// Creating info text with a little history of what happened in the station for debugging purpose		
			strInfo := fbHistoryInfo.CreateStationInfo(nStationIndex, nMoverIndex, nNextStationIndex);	
			
				// Move on track command	
				GVL.g_Movers[nMoverIndex].std.MoveOnTrackExt('move on track', GVL.g_Tracks[nTrackIndex].std, fMoverToTrackPosition,
 								fMoverVelocity, fMoverAcceleration , fMoverJerk, stMoveOnTrackParameters);											 
			
			
			nStateProcess := nStateProcess +1;
			
		
		
	131: 	// Checking move command return
			IF GVL.g_Movers[nMoverIndex].std.P_MoveOnTrackExt.Active
			OR GVL.g_Movers[nMoverIndex].std.P_MoveOnTrackExt.Done 
			THEN
				nStateProcess := 200;
				
			ELSIF GVL.g_Movers[nMoverIndex].std.P_MoveOnTrackExt.Error THEN
				   nErrorID := GVL.g_Movers[nMoverIndex].std.P_MoveOnTrackExt.ErrorID;
				  nObjectID := GVL.g_Movers[nMoverIndex].std.P_MoveOnTrackExt.stInfo.nObjectID;
				nObjectType := GVL.g_Movers[nMoverIndex].std.P_MoveOnTrackExt.stInfo.nObjectType;
			END_IF		
			
	200: // send mover to load position 
			loadPosition.SetValuesXY(650,180);
	
	
		IF NOT GVL.g_Movers[nMoverIndex].std.P_Busy THEN
			stMoveToPositionOptions.useOrientation := TRUE;
			GVL.g_Movers[nMoverIndex].std.MoveToPositionExt(strInfo, loadPosition, 100, 1000, 1000, 1000, stMoveToPositionOptions);
			nStateProcess := nStateProcess +1;
		END_IF
		
	201: //check state 
			
		IF GVL.g_Movers[nMoverIndex].std.P_MoveToPositionExt.Done THEN
				nStateProcess := nStateProcess +9;
			ELSIF GVL.g_Movers[nMoverIndex].std.P_MoveToPositionExt.Error THEN
				   nErrorID := GVL.g_Movers[nMoverIndex].std.P_MoveToPositionExt.ErrorID;
				  nObjectID := GVL.g_Movers[nMoverIndex].std.P_MoveToPositionExt.stInfo.nObjectID;
				nObjectType := GVL.g_Movers[nMoverIndex].std.P_MoveToPositionExt.stInfo.nObjectType;
		END_IF
			
		//	GVL.g_Stations[GVL.PuncherSeparateStation].P_ProcessState:= ST_EStationProcessState.Empty;

	210:  // wait for signal to load part 
			//IF  GVL.g_Stations[GVL.PuncherStation].P_ProcessRequest:=GVL.PuncherSeparateStation THEN 
				
			//	GVL.g_Stations[GVL.PuncherSeparateStation].P_ProcessState:= ST_EStationProcessState.InProcess;
				nStateProcess := nStateProcess +1;
				
		//	END_IF
		
	211: // command grab part 
			IF NOT bPartInGripper THEN 
				// cmd grab part 
				nStateProcess := nStateProcess +1;
			END_IF
	212: //check gripper sensors
		
		//if sensor= true then 
				bPartInGripper:=TRUE;
				nStateProcess := nStateProcess +1;
				
				
	213: //go to rotate position 
		 // send mover to load position 
			rotatePosition.SetValuesXY(600,180);
	
	
		IF NOT GVL.g_Movers[nMoverIndex].std.P_Busy THEN
			stMoveToPositionOptions.useOrientation := TRUE;
			GVL.g_Movers[nMoverIndex].std.MoveToPositionExt(strInfo, rotatePosition, 100, 1000, 1000, 1000, stMoveToPositionOptions);
			nStateProcess := nStateProcess +1;
		END_IF
		
	214: //check state 
			
		IF GVL.g_Movers[nMoverIndex].std.P_MoveToPositionExt.Done THEN
				nStateProcess := nStateProcess +7;
			ELSIF GVL.g_Movers[nMoverIndex].std.P_MoveToPositionExt.Error THEN
				   nErrorID := GVL.g_Movers[nMoverIndex].std.P_MoveToPositionExt.ErrorID;
				  nObjectID := GVL.g_Movers[nMoverIndex].std.P_MoveToPositionExt.stInfo.nObjectID;
				nObjectType := GVL.g_Movers[nMoverIndex].std.P_MoveToPositionExt.stInfo.nObjectType;
		END_IF

	
	
	
	

	215://  rotate 90 degrees
	
			fSendAwayPosition		:=50;	
			fMoverToTrackPosition := fSendAwayPosition;
			nTrackIndex           := nStationTrackIndex;
			fMoverVelocity     	  :=    300.0;
			fMoverAcceleration 	  :=  1_000.0;
			fMoverJerk         	  := 10_000.0;	
	
			stMoveRotateOptions.direction := Tc3_Mc3PlanarMotion.MC_DIRECTION.mcDirectionPositive;	

			
			// Creating info text with a little history of what happened in the station for debugging purpose		
			strInfo := fbHistoryInfo.CreateStationInfo(nStationIndex, nMoverIndex, nNextStationIndex);	
			
				// Move on track command	
										 
			GVL.g_Movers[nMoverIndex].std.MoveC('rotate ',90, fMoverToTrackPosition,
 								fMoverVelocity, fMoverAcceleration , fMoverJerk, stMoveRotateOptions);
			
			nStateProcess := nStateProcess +1;
			
	216: 		//join track 
	
		IF NOT GVL.g_Movers[nMoverIndex].std.P_Busy THEN
			stJoinTrackOptions.useOrientation := FALSE;
			GVL.g_Movers[nMoverIndex].std.JoinTrack(strInfo, GVL.g_Tracks[nTrackIndex].std, 100, 1000, 1000, stJoinTrackOptions);
			
			nStateProcess := nStateProcess +1;
		END_IF
	217:
		IF GVL.g_Movers[nMoverIndex].std.P_JoinTrack.Done THEN
			gvl.g_Movers[nMoverIndex].P_TrackId:=nTrackIndex;
			nStateProcess := nStateProcess+1;
		ELSIF GVL.g_Movers[nMoverIndex].std.P_JoinTrack.Error THEN
			   nErrorID := GVL.g_Movers[nMoverIndex].std.P_JoinTrack.ErrorID;
			  nObjectID := GVL.g_Movers[nMoverIndex].std.P_JoinTrack.stInfo.nObjectID;
			nObjectType := GVL.g_Movers[nMoverIndex].std.P_JoinTrack.stInfo.nObjectType;
		END_IF	
	
		
	218: 	// Checking move command return
			IF GVL.g_Movers[nMoverIndex].std.P_MoveC.Active
			OR GVL.g_Movers[nMoverIndex].std.P_MoveC.Done 
			THEN
				nStateProcess := nStateProcess + 1;
				
			ELSIF GVL.g_Movers[nMoverIndex].std.P_MoveC.Error THEN
				   nErrorID := GVL.g_Movers[nMoverIndex].std.P_MoveC.ErrorID;
				  nObjectID := GVL.g_Movers[nMoverIndex].std.P_MoveC.stInfo.nObjectID;
				nObjectType := GVL.g_Movers[nMoverIndex].std.P_MoveC.stInfo.nObjectType;
			END_IF	
	
	219:// move forward to camera 
	
			fSendAwayPosition		:=50;	
			fMoverToTrackPosition := fSendAwayPosition;
			nTrackIndex           := nStationTrackIndex;
			fMoverVelocity     	  :=    300.0;
			fMoverAcceleration 	  :=  1_000.0;
			fMoverJerk         	  := 10_000.0;	
	
			stMoveOnTrackParameters.direction := Tc3_Mc3PlanarMotion.MC_DIRECTION.mcDirectionShortestWay;	
			stMoveOnTrackParameters.gap := 120.0;

			
			// Creating info text with a little history of what happened in the station for debugging purpose		
			strInfo := fbHistoryInfo.CreateStationInfo(nStationIndex, nMoverIndex, nNextStationIndex);	
			
				// Move on track command	
			GVL.g_Movers[nMoverIndex].std.MoveOnTrackExt('move on track', GVL.g_Tracks[nTrackIndex].std, fMoverToTrackPosition,
 								fMoverVelocity, fMoverAcceleration , fMoverJerk, stMoveOnTrackParameters);											 
			
			
			nStateProcess := nStateProcess +1;
			
		
		
	220: 	// Checking move command return
			IF GVL.g_Movers[nMoverIndex].std.P_MoveOnTrackExt.Active
			OR GVL.g_Movers[nMoverIndex].std.P_MoveOnTrackExt.Done 
			THEN
				nStateProcess := nStateProcess + 2;
				
			ELSIF GVL.g_Movers[nMoverIndex].std.P_MoveOnTrackExt.Error THEN
				   nErrorID := GVL.g_Movers[nMoverIndex].std.P_MoveOnTrackExt.ErrorID;
				  nObjectID := GVL.g_Movers[nMoverIndex].std.P_MoveOnTrackExt.stInfo.nObjectID;
				nObjectType := GVL.g_Movers[nMoverIndex].std.P_MoveOnTrackExt.stInfo.nObjectType;
			END_IF	
	
// 
// 	221: 	// on camera position handshake
// 
// 			GVL.g_Stations[GVL.PuncherSeparateStation].P_ProcessRequest:= CMD_CameraCheck; 
// wait for camera feedback 
// 			IF THIS^.bCameraProcessDone THEN 
// 				nStateProcess := nStateProcess + 1;
// 				THIS^.bCMD_CameraCheck:=FALSE; 
// 			END_IF
// 				
		
	222:	// move forward to pucher 
			fSendAwayPosition		:=80;	
			fMoverToTrackPosition := fSendAwayPosition;
			nTrackIndex           := nStationTrackIndex;
			fMoverVelocity     	  :=    300.0;
			fMoverAcceleration 	  :=  1_000.0;
			fMoverJerk         	  := 10_000.0;	
	
			stMoveOnTrackParameters.direction := Tc3_Mc3PlanarMotion.MC_DIRECTION.mcDirectionShortestWay;	
			stMoveOnTrackParameters.gap       := 120.0;

			
			// Creating info text with a little history of what happened in the station for debugging purpose		
			strInfo := fbHistoryInfo.CreateStationInfo(nStationIndex, nMoverIndex, nNextStationIndex);	
			
				// Move on track command	
			GVL.g_Movers[nMoverIndex].std.MoveOnTrackExt('move on track', GVL.g_Tracks[nTrackIndex].std, fMoverToTrackPosition,
 								fMoverVelocity, fMoverAcceleration , fMoverJerk, stMoveOnTrackParameters);											 
			
			
			nStateProcess := nStateProcess +1;
			
		
		
	223: 	// Checking move command return
			IF GVL.g_Movers[nMoverIndex].std.P_MoveOnTrackExt.Active
			OR GVL.g_Movers[nMoverIndex].std.P_MoveOnTrackExt.Done 
			THEN
				nStateProcess := nStateProcess + 1;
				
			ELSIF GVL.g_Movers[nMoverIndex].std.P_MoveOnTrackExt.Error THEN
				   nErrorID := GVL.g_Movers[nMoverIndex].std.P_MoveOnTrackExt.ErrorID;
				  nObjectID := GVL.g_Movers[nMoverIndex].std.P_MoveOnTrackExt.stInfo.nObjectID;
				nObjectType := GVL.g_Movers[nMoverIndex].std.P_MoveOnTrackExt.stInfo.nObjectType;
			END_IF	

	
	224:
			// check sensors  puncher gripper 
			nStateProcess := nStateProcess + 1;
			
	225: // move back 
	
			fSendAwayPosition		:=0;	
			fMoverToTrackPosition := fSendAwayPosition;
			nTrackIndex           := nStationTrackIndex;
			fMoverVelocity     	  :=    300.0;
			fMoverAcceleration 	  :=  1_000.0;
			fMoverJerk         	  := 10_000.0;	
	
			stMoveOnTrackParameters.direction := Tc3_Mc3PlanarMotion.MC_DIRECTION.mcDirectionShortestWay;	
			stMoveOnTrackParameters.gap       := 120.0;

			
			// Creating info text with a little history of what happened in the station for debugging purpose		
			strInfo := fbHistoryInfo.CreateStationInfo(nStationIndex, nMoverIndex, nNextStationIndex);	
			
				// Move on track command	
			GVL.g_Movers[nMoverIndex].std.MoveOnTrackExt('move on track', GVL.g_Tracks[nTrackIndex].std, fMoverToTrackPosition,
 								fMoverVelocity, fMoverAcceleration , fMoverJerk, stMoveOnTrackParameters);											 
			
			
			nStateProcess := nStateProcess +1;
			
		
		
	226: 	// Checking move command return
			IF GVL.g_Movers[nMoverIndex].std.P_MoveOnTrackExt.Active
			OR GVL.g_Movers[nMoverIndex].std.P_MoveOnTrackExt.Done 
			THEN
				nStateProcess := nStateProcess + 1;
				
			ELSIF GVL.g_Movers[nMoverIndex].std.P_MoveOnTrackExt.Error THEN
				   nErrorID := GVL.g_Movers[nMoverIndex].std.P_MoveOnTrackExt.ErrorID;
				  nObjectID := GVL.g_Movers[nMoverIndex].std.P_MoveOnTrackExt.stInfo.nObjectID;
				nObjectType := GVL.g_Movers[nMoverIndex].std.P_MoveOnTrackExt.stInfo.nObjectType;
			END_IF	
	
	227://  rotate 90 degrees
	
			fSendAwayPosition		:=50;	
			fMoverToTrackPosition := fSendAwayPosition;
			nTrackIndex           := nStationTrackIndex;
			fMoverVelocity     	  :=    300.0;
			fMoverAcceleration 	  :=  1_000.0;
			fMoverJerk         	  := 10_000.0;	
	
			stMoveRotateOptions.direction := Tc3_Mc3PlanarMotion.MC_DIRECTION.mcDirectionPositive;	

			
			// Creating info text with a little history of what happened in the station for debugging purpose		
			strInfo := fbHistoryInfo.CreateStationInfo(nStationIndex, nMoverIndex, nNextStationIndex);	
			
				// Move on track command	
										 
			GVL.g_Movers[nMoverIndex].std.MoveC('rotate',90, fMoverToTrackPosition,
 								fMoverVelocity, fMoverAcceleration , fMoverJerk, stMoveRotateOptions);
			
			nStateProcess := nStateProcess +1;
			
		
		
	228: 	// Checking move command return
			IF GVL.g_Movers[nMoverIndex].std.P_MoveC.Active
			OR GVL.g_Movers[nMoverIndex].std.P_MoveC.Done 
			THEN
				nStateProcess := 500;
				
			ELSIF GVL.g_Movers[nMoverIndex].std.P_MoveC.Error THEN
				   nErrorID := GVL.g_Movers[nMoverIndex].std.P_MoveC.ErrorID;
				  nObjectID := GVL.g_Movers[nMoverIndex].std.P_MoveC.stInfo.nObjectID;
				nObjectType := GVL.g_Movers[nMoverIndex].std.P_MoveC.stInfo.nObjectType;
			END_IF	
	
	
	
	500: 	// Done for this cycle
		//	GVL.g_Stations[GVL.PuncherSeparateStation].P_ProcessState:=ST_EStationProcessState.Finished;
		IF 	GVL.g_Stations[GVL.PuncherStation].P_ProcessRequest<>GVL.PuncherSeparateStation THEN 
				nStateProcess := 200;
		END_IF 

END_CASE
END_METHOD

END_FUNCTION_BLOCK

// ---- Stations/Base/FB_StationBase.TcPOU
FUNCTION_BLOCK FB_StationBase IMPLEMENTS I_Station


VAR
	stMoveOnTrackParameters 	: ST_MoveOnTrackOptions; 
	stMoveRotateOptions	: ST_MoveCOptions; 	
	stStationPosition	: ST_StationPosition;	
	eProcessMode		: E_ProcessMode;
	StationPosition     : PositionXYC;	
	stMoveToPositionOptions: ST_MoveToPositionOptions;
	stJoinTrackOptions: ST_JoinTrackOptions;
	stLeaveTrackOptions: ST_LeaveTrackOptions;
	
	idx  				: UDINT;
	nStateInit			: UDINT;
	nStateClear 		: UDINT;
	nStateProcess		: UDINT;
	bStationInitDone	: BOOL;	
	
	
	// Lists for Stations
	fbList_Station		: FB_List;
	fbList_InputW		: FB_List;		
	fbList_InputS		: FB_List;	
	fbList_InputE		: FB_List;		
	fbList_InputN		: FB_List;	
	
	// History info for debugging purpose
	strInfo				: STRING;	
	fbHistoryInfo		: FB_HistoryInfo;	
	
	
	nProcessRequest		: DINT;
	nProcessClearence	: DINT;
	nProcessState		: DINT;
	
	fStationPositionOnTrack		: LREAL;	
	
	// =========================
	nStationIndex				: UINT;
	
	nPreviousStationIndexInputW : UINT;	
	nTrackIndexInputW 			: UINT;		
	nPreviousStationIndexInputS : UINT;	
	nTrackIndexInputS 			: UINT;		
	nPreviousStationIndexInputE : UINT;	
	nTrackIndexInputE 			: UINT;		
	nPreviousStationIndexInputN : UINT;	
	nTrackIndexInputN 			: UINT;		
	
	nNextStationIndexOutputW 	: UINT;	
	nTrackIndexOutputW 			: UINT;		
	nNextStationIndexOutputS 	: UINT;	
	nTrackIndexOutputS 			: UINT;		
	nNextStationIndexOutputE 	: UINT;	
	nTrackIndexOutputE 			: UINT;		
	nNextStationIndexOutputN 	: UINT;	
	nTrackIndexOutputN 			: UINT;
	
	fStationPosition_X 			: LREAL;
	fStationPosition_Y 			: LREAL;
	fInRangeDistance			: LREAL;	
	
	fSendAwayDistanceOutputW    : LREAL;	  
    fSendAwayDistanceOutputS    : LREAL;
	fSendAwayDistanceOutputE    : LREAL;	
	fSendAwayDistanceOutputN    : LREAL;
	
	fSendAwayPositionOutputW	: LREAL;
	fSendAwayPositionOutputS	: LREAL;
	fSendAwayPositionOutputE	: LREAL;
	fSendAwayPositionOutputN	: LREAL;	
	
	nStationTrackIndex			: UINT;
	nStationTaskList              :ARRAY[1..200] OF  UDINT; 

	position					: PositionXYC;
END_VAR

METHOD Clear : BOOL
VAR_INPUT
END_VAR


VAR_INST

	nStateClear : UINT;

END_VAR


	CASE nStateClear OF 
		
	0:	// Enter
		            Clear := FALSE;
		  nProcessRequest := 0;
		nProcessClearence := 0;
		    nProcessState := 0;	  
			  
		nStateClear := nStateClear +10;
		
	10: // Clear Station-List
		IF fbList_Station.ClearList() THEN
			nStateClear := nStateClear +10;	
		END_IF
		
	20: // Clear InputW-List
		IF fbList_InputW.ClearList() THEN
			nStateClear := nStateClear +10;	
		END_IF
	
	30: // Clear InputE-List
		IF fbList_InputE.ClearList() THEN
			nStateClear := nStateClear +10;	
		END_IF	
	
	40: // Clear InputS-List
		IF fbList_InputS.ClearList() THEN
			nStateClear := nStateClear +10;	
		END_IF		
	
	50: // Clear InputN-List
		IF fbList_InputN.ClearList() THEN
			nStateClear := nStateClear +10;	
		END_IF
	
	60:	nStateClear := 100;	
		
		
	100:  // Done
		nStateClear := 0;
		      Clear := TRUE;
		
	END_CASE
END_METHOD

METHOD Cycle : BOOL
VAR_INPUT
END_VAR
VAR
	nForCounter : INT;
END_VAR


VAR_INST
	
	fTestValueX	: LREAL;
	fTestValueY : LREAL;	
	
END_VAR
;
END_METHOD

METHOD Init : BOOL


	  nStateInit := 0;
	nStateProcess := 0;
	 eProcessMode := E_ProcessMode.None;

	Init := TRUE;
END_METHOD

PROPERTY P_bInitDone : BOOL
GET
P_bInitDone := bStationInitDone;
END_GET
END_PROPERTY

PROPERTY P_eProcessMode : E_ProcessMode
GET
P_eProcessMode := eProcessMode;
END_GET
SET
eProcessMode := P_eProcessMode;
END_SET
END_PROPERTY

PROPERTY P_List_Station : I_List
GET
P_List_Station := fbList_Station;
END_GET
END_PROPERTY

PROPERTY P_List_Switch_Input_E : I_List
GET
P_List_Switch_Input_E := fbList_InputE;
END_GET
END_PROPERTY

{warning 'Add property implementation'}
PROPERTY P_List_Switch_Input_N : I_List
GET
P_List_Switch_Input_N := fbList_InputN;
END_GET
END_PROPERTY

PROPERTY P_List_Switch_Input_S : I_List
GET
P_List_Switch_Input_S := fbList_InputS;
END_GET
END_PROPERTY

PROPERTY P_List_Switch_Input_W : I_List
GET
P_List_Switch_Input_W := fbList_InputW;
END_GET
END_PROPERTY

PROPERTY P_nErrorCode : UDINT
GET
END_GET
END_PROPERTY

PROPERTY P_Position : ST_StationPosition
GET
P_Position := stStationPosition;
END_GET
END_PROPERTY

PROPERTY P_ProcessClearance : DINT
GET
P_ProcessClearance := nProcessClearence;
END_GET
END_PROPERTY

PROPERTY P_ProcessRequest : UDINT
GET
P_ProcessRequest := nProcessRequest;
END_GET
SET
nProcessRequest := P_ProcessRequest;
END_SET
END_PROPERTY

PROPERTY P_ProcessState : UDINT
GET
P_ProcessState := nProcessState;
END_GET
SET
nProcessState := P_ProcessState;
END_SET
END_PROPERTY

PROPERTY P_StationTaskList : array[1..200] of UDINT
GET
 P_StationTaskList := nStationTaskList;
END_GET
SET
nStationTaskList := P_StationTaskList;
END_SET
END_PROPERTY

METHOD Process : BOOL
END_METHOD

END_FUNCTION_BLOCK

// ---- Stations/Helper/FB_HistoryInfo.TcPOU
FUNCTION_BLOCK FB_HistoryInfo


VAR
	strInfo				: STRING;
	strInfoHistory		: ARRAY[0..10] OF STRING;
END_VAR

METHOD AddEntry : BOOL
VAR_INPUT
	sInfo	: STRING;
END_VAR


VAR
	idx	: UDINT;
END_VAR


	FOR idx:=10 TO 1 BY -1 DO 
		strInfoHistory[idx] := strInfoHistory[idx-1];
	END_FOR
	strInfoHistory[0] := sInfo;
END_METHOD

METHOD CreateStationInfo : STRING
VAR_INPUT
	nStationIndex		: UDINT;
	nMoverIndex			: UDINT;
	nNextStationIndex   : UDINT;
END_VAR



VAR
	strInfo			: STRING;	
END_VAR


	strInfo := CONCAT('St:', UDINT_TO_STRING(nStationIndex));
	strInfo := CONCAT(strInfo, ' M:');
	strInfo := CONCAT(strInfo, UDINT_TO_STRING(nMoverIndex));
	strInfo := CONCAT(strInfo, ' to next station:');
	strInfo := CONCAT(strInfo, UDINT_TO_STRING(nNextStationIndex));
	
	CreateStationInfo := strInfo;		
			
	THIS^.AddEntry(strInfo);
END_METHOD

END_FUNCTION_BLOCK

// ---- Stations/FB_PuncherBufferStation.TcPOU
FUNCTION_BLOCK FB_PuncherBufferStation EXTENDS FB_StationBase

METHOD Clear : BOOL
	CASE nStateClear OF
		
	0:	// Enter
		Clear := FALSE;
		nStateClear := nStateClear +10;
		
	10: // Clearing all Station-Lists 
		IF SUPER^.Clear() THEN
			nStateClear := nStateClear +10;
		END_IF	
	
	20:	// Add aditional Data to be cleared here...
		nStateClear := 100;
		
		
	100: // Done
		      Clear := TRUE;
		nStateClear := 0;

	END_CASE
END_METHOD

METHOD Init : BOOL


VAR_INST
	nTestCounter	: INT;	
END_VAR
nTestCounter := nTestCounter +1;

CASE nStateInit OF

	0:		// Enter 
			bStationInitDone := FALSE;
			   nStateProcess := 0;
			      nStateInit := 10;
				 
			
	10:		// Init Station-Parameters				
				  nStationIndex := 3;				// Each station needs an unique index	
			 nStationTrackIndex := 4;	 			// Track on which the station resides
			 
			 
	nPreviousStationIndexInputW := 7;
			  nTrackIndexInputW := 10;
	   nNextStationIndexOutputW := 1;
	   		 nTrackIndexOutputW := 1;	 
			 
			 
			 	  
			 fStationPosition_X := 660.0;			// Position of the station in X/Y coordinates
			 fStationPosition_Y := 420.0;			// Position of the station in X/Y coordinates
			  
	   fSendAwayDistanceOutputW := 300.0;
	   fSendAwayDistanceOutputN := 100.0;			// Position on track a mover will be send to after processing 
			  fInRangeDistance  := 300.0;			// Position in front of a station from where a mover will be taken over
			  
			  nStateInit := 11;
				   
				  
	11: // Fail-safe check, just to make sure all variables have been assigned after doing copy&paste from the template
			IF        nStationIndex > 0
			AND  nStationTrackIndex > 0
			AND  nPreviousStationIndexInputW > 0
			AND  nTrackIndexInputW > 0
			AND  nNextStationIndexOutputW > 0
			AND  nTrackIndexOutputW > 0
			AND  fStationPosition_X > 0
			AND  fStationPosition_Y > 0
			AND  fSendAwayDistanceOutputW <> 0
			AND   fInRangeDistance > 0
			THEN   
				nStateInit := 20;
			END_IF
			
				   
	20:		// Calculating positions
	
			// 1. Calculating station position on track
			position.SetValuesXYC(fStationPosition_X, fStationPosition_Y, 0.0);
			//fStationPositionOnTrack := GVL.g_Tracks[nStationTrackIndex].std.GetTrackPositionAt_XY(fStationPosition_X, fStationPosition_Y);
			fStationPositionOnTrack := GVL.g_Tracks[nStationTrackIndex].P_TrackLength;;
							
			// 2. Calculating send-away position on track
			fSendAwayPositionOutputW := fStationPositionOnTrack + fSendAwayDistanceOutputW; 
			
			// The send away position must not exceed the lenght of the track!
			IF fSendAwayPositionOutputW > GVL.g_Tracks[nStationTrackIndex].P_TrackLength THEN
				fSendAwayPositionOutputW := GVL.g_Tracks[nStationTrackIndex].P_TrackLength;
			END_IF
			
			// 3. Calculating the station position in X/Y coordinates determined by the track	
            //    This is to make sure the center of the station is always located directly on the track.
			//    This value can differ from the initial fStationPosition_X, fStationPosition_Y in case they were not matching the track
			GVL.g_Tracks[nStationTrackIndex].std.GetMoverPositionAt(fStationPositionOnTrack, StationPosition);
			
			// Providing the station position to e.g. visualization	
			stStationPosition.bInit            := TRUE;
			stStationPosition.fPositionOnTrack := fStationPositionOnTrack;
			stStationPosition.nTrackId         := nStationTrackIndex;
			stStationPosition.fPosition_X	   := StationPosition.x;
			stStationPosition.fPosition_Y	   := StationPosition.y;

			nStateInit := 30;
			
			
	30:		// Clear Lists
			IF THIS^.Clear() THEN
				nStateInit := 90;	
			END_IF

			
		
	90:		// Creating a little history of what happened in the station for debugging purpose
			fbHistoryInfo.AddEntry('Init');
	
			nStateInit := 100;
			
						
	100:	// Init done
			IF SUPER^.Init() THEN
				bStationInitDone := TRUE;	
				           Init := TRUE;
			END_IF
				
	
END_CASE
END_METHOD

METHOD Process : BOOL

VAR_INST
		
	nMoverIndex				: UINT;
	(*
	fMoverToTrackPosition	: LREAL;
	nTrackIndex				: UINT;
	fMoverVelocity			: LREAL;
	fMoverAcceleration		: LREAL;
	fMoverJerk				: LREAL;
	
	
	nErrorId				: UDINT;
	nObjectID				: UDINT;
	nObjectType				: UDINT;		
	
	
	// Process
	nDestinationProcess		: UINT;
	nIncommingTrackOID		: UDINT;
	nNextStationIndex		: UINT;		 				
	fSendAwayPosition		: LREAL;
	nTrackindexNext			: UINT;
	*)
	
END_VAR
// Station - Switch-Seperate

CASE nStateProcess OF 

	0:		// Enter
			IF bStationInitDone THEN
				nStateProcess := 100;
			END_IF

	
	100: 	// Waiting for Mover
			IF P_List_Switch_Input_W.P_FirstInList <> 0 THEN
				P_List_Station.AddMover(P_List_Switch_Input_W.RemoveFirstInList());
			    nStateProcess := nStateProcess +10;
			END_IF
	
			
	110:	// Working with the station list from here on	
			IF P_List_Station.P_FirstInList <> 0 THEN
				nMoverIndex := P_List_Station.P_FirstInList.P_Id;
			    nStateProcess := nStateProcess +10;
			END_IF		
			
		
	120: 	// Check if Mover is in range
			IF  GVL.g_Movers[nMoverIndex].std.P_SetOnTrack.TrackOID = GVL.g_Tracks[nTrackIndexInputW].std.P_OID
			AND GVL.g_Movers[nMoverIndex].std.P_SetOnTrack.SetPos   > fStationPositionOnTrack - fInRangeDistance
			THEN
				nStateProcess := nStateProcess +10;
			END_IF
			
			
// 			
// 	130: // Decide to which Station the mover has to travel to next.	
// 			IF 	GVL.g_Stations[PuncherStation].P_ProcessState
// 				
// 				// -> Wait in buffer 
// 				nNextStationIndex  := nNextStationIndexOutputB;
// 				fSendAwayPosition  := fSendAwayPositionOutputB;
// 				nTrackindexNext    := nTrackIndexOutputB;		
// 		
// 			ELSE: // -> send to puncher
// 				nNextStationIndex  := nNextStationIndexOutputC;
// 				fSendAwayPosition  := fSendAwayPositionOutputC;
// 				nTrackindexNext    := nTrackIndexOutputC;				
// 		END_IF
// 			
// 				nStateProcess := 200;	
// 		
// 			
// 			
// 		
// 	200: 	// Send mover to the next station	
// 			fMoverToTrackPosition := fSendAwayPosition;
// 			nTrackIndex           := nTrackindexNext;
// 			fMoverVelocity     	  :=    300.0;
// 			fMoverAcceleration 	  :=  1_000.0;
// 			fMoverJerk         	  := 10_000.0;	
// 	
// 			stMoveParameters.direction := Tc3_Mc3PlanarMotion.MC_DIRECTION.mcDirectionPositive;	
// 			stMoveParameters.gap       := 240.0;
// 
// 			
// 			// Creating info text with a little history of what happened in the station for debugging purpose		
// 			strInfo := fbHistoryInfo.CreateStationInfo(nStationIndex, nMoverIndex, nNextStationIndex);	
// 			
// 				
// 			// Move on track command	
// 			ipMoverApplication[nMoverIndex].std.MoveOnTrack( strInfo,
// 															 ipTrack[nTrackIndex].std,
// 															 fMoverToTrackPosition,
// 															 fMoverVelocity,
// 															 fMoverAcceleration,
// 															 fMoverJerk,
// 															 stMoveParameters.gap,
// 															 stMoveParameters.direction);
// 			nStateProcess := nStateProcess +1;
// 			
// 		
// 		
// 	201: 	// Checking move command return
// 			IF ipMoverApplication[nMoverIndex].std.P_MoveOnTrack.Active
// 			OR ipMoverApplication[nMoverIndex].std.P_MoveOnTrack.Done 
// 			THEN
// 				nStateProcess := nStateProcess + 9;
// 				
// 			ELSIF ipMoverApplication[nMoverIndex].std.P_MoveOnTrack.Error THEN
// 				   nErrorID := ipMoverApplication[nMoverIndex].std.P_MoveOnTrack.ErrorID;
// 				  nObjectID := ipMoverApplication[nMoverIndex].std.P_MoveOnTrack.stInfo.nObjectID;
// 				nObjectType := ipMoverApplication[nMoverIndex].std.P_MoveOnTrack.stInfo.nObjectType;
// 			END_IF		
// 		
// 	
// 	210:	// Wait till the mover passed the junction point
// 			IF ipMoverApplication[nMoverIndex].std.P_SetOnTrack.TrackOID <> ipTrack[nTrackIndexInputA].std.P_OID THEN
// 				nStateProcess := nStateProcess + 10;
// 			END_IF		
// 
// 		
// 	220: 	// Mover to the list of the next station
// 			ipStation[nNextStationIndex].P_List_Station.AddMover(P_List_Station.RemoveFirstInList());
// 			nStateProcess := 500;	
// 	*)
// 		
// 	500: 	// Done for this cycle
// 			nStateProcess := 100;

END_CASE
END_METHOD

END_FUNCTION_BLOCK
